Universal Robots PolyScope program: taskboard_belt_v7.urp

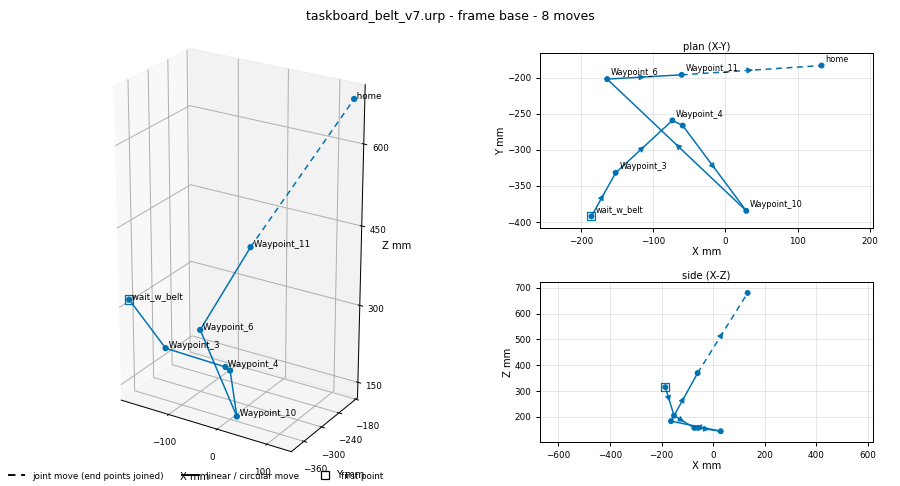
[picture p0: tool path of taskboard_belt_v7.urp in frame base, 8 of 9 moves have a stored position in this frame; points joined in program order, loops and branches not executed]
Program taskboard_belt_v7 (installation=default directory=/programs/wrs2020 createdIn=5.6.0.90886 lastSavedIn=5.9.1.1031110 robotSerialNumber=20205500180)
Calibrated DH parameters: a=[0, -0.425, -0.3922, 0, 0, 0]; d=[0.1625, 0, 0, 0.1333, 0.0997, 0.0996]; alpha=[1.570796, 0, 0, 1.570796, -1.570796, 0]; deltaTheta=[0, 0, 0, 0, 0, 0]
Robot Program (runOnlyOnce=true)
  MoveJ speed 60 deg/s, acceleration 80 deg/s^2 (useActiveTCP=true) feature=Base
    currentpose := get_actual_joint_positions()
    Waypoint Waypoint (Variable): variable=currentpose
  SuppressedNode
    Folder pick blind
      MoveJ speed 120 deg/s, acceleration 120 deg/s^2 (useActiveTCP=false) tcp=TCP; feature=Base
        Waypoint home: TCP in base x=132.399 y=-179.474 z=460.725 mm, rx=-0.0051 ry=-3.1414 rz=-0.0307 rad; joints [89.952, -120.316, 80.22, -48.701, -89.95, -0.003] deg; TCP offset x=0 y=0 z=220 mm, rx=0 ry=0 rz=0 rad
        Waypoint Waypoint_12: TCP in base x=-118.553 y=-294.346 z=577.587 mm, rx=1.3176 ry=2.7241 rz=-0.2718 rad; joints [40.024, -118.444, 99.589, -78.038, -80.282, 2.128] deg
      URCap Gripper (Robotiq_Grippers, Robotiq Inc.) dataModel(position=48.23529411764706, force=100.0, speed=100.0, positionInDouble=48.23529411764706, forceInDouble=100.0, speedInDouble=100.0, slaveIds=[9], blocking=true)
      MoveJ speed 120 deg/s, acceleration 100 deg/s^2 (useActiveTCP=false) tcp=TCP; feature=Base
        Waypoint Waypoint_1: TCP in base x=-147.509 y=-481.576 z=322.425 mm, rx=-2.2532 ry=2.177 rz=0.038 rad; joints [57.916, -85.82, 110.34, -113.684, -91.081, -124] deg; TCP offset x=0 y=0 z=0 mm, rx=0 ry=0 rz=0 rad
        MoveL speed 100 mm/s, acceleration 1200 mm/s^2 (useActiveTCP=false) tcp=TCP; feature=Base
          Waypoint Waypoint_2: TCP in base x=-147.509 y=-481.576 z=273.212 mm, rx=2.2507 ry=-2.1796 rz=-0.0127 rad; joints [57.763, -82.536, 115.155, -122.915, -90.37, -124] deg; TCP offset x=0 y=0 z=0 mm, rx=0 ry=0 rz=0 rad
      URCap Gripper (Robotiq_Grippers, Robotiq Inc.) dataModel(position=100.0, force=100.0, speed=100.0, positionInDouble=100.0, forceInDouble=100.0, speedInDouble=100.0, slaveIds=[9], blocking=true)
      MoveL speed 250 mm/s, acceleration 1200 mm/s^2 (useActiveTCP=true) feature=Base
        MoveDirectionNode (selectedDirection=ZPlus)
          Until DISTANCE (allowActions=false deceleration=3 distanceNodeType=STOP) Distance=0.1; motionParameters(blendRadius=0)
  MoveL speed 800 mm/s, acceleration 400 mm/s^2 (useActiveTCP=false) tcp=TCP; feature=Base
    SuppressedNode
      Waypoint above_tray: motionParameters(blendRadius=0.05); TCP in base x=-172.311 y=-492.624 z=406.821 mm, rx=2.0826 ry=-2.3042 rz=0.0252 rad; joints [55.84, -87.577, 100.035, -104.661, -89.581, -118.368] deg
    Waypoint wait_w_belt: TCP in base x=-185.572 y=-392.078 z=315.254 mm, rx=-1.4441 ry=1.9502 rz=-1.0486 rad; joints [37.028, -91.796, 114.934, -76.388, -46.414, -141.19] deg
  Popup Message (haltProgram=false message=start sequence together with b_bot (simultaneous start) inputType=Text)
  MoveL speed 500 mm/s, acceleration 1200 mm/s^2 (useActiveTCP=false) tcp=TCP; feature=Base
    SuppressedNode
      Waypoint Waypoint_5: TCP in base x=-173.43 y=-369.039 z=261.712 mm, rx=-1.282 ry=1.8047 rz=-1.1483 rad; joints [34.616, -88.409, 119.828, -68.558, -43.225, -150.47] deg
    Waypoint Waypoint_3: motionParameters(blendRadius=0.05); TCP in base x=-152.025 y=-331.758 z=204.759 mm, rx=-0.9043 ry=1.7298 rz=-1.6658 rad; joints [27.571, -85.137, 129.926, -53.568, -24.794, -175.111] deg
    Waypoint Waypoint_4: motionParameters(blendRadius=0.01); TCP in base x=-73.392 y=-259.129 z=157.442 mm, rx=-0.7441 ry=1.8696 rz=-1.7976 rad; joints [17.552, -96.937, 152.26, -63.92, -23.073, -175.094] deg
    Waypoint Waypoint_9: TCP in base x=-59.125 y=-266.29 z=157.434 mm, rx=-0.7441 ry=1.8696 rz=-1.7976 rad; joints [21.298, -97.571, 152.76, -64.841, -19.306, -173.924] deg
    SuppressedNode
      Waypoint Waypoint_7: TCP in base x=-93.501 y=-273.032 z=162.831 mm, rx=-0.9044 ry=1.7298 rz=-1.6658 rad; joints [21.869, -90.172, 144.622, -61.38, -30.363, -177.16] deg
  Wait Sleep waitTime=10
  URCap Gripper (Robotiq_Grippers, Robotiq Inc.) dataModel(position=80.3921568627451, force=0.0, speed=0.0, positionInDouble=80.3921568627451, forceInDouble=0.0, speedInDouble=0.0, slaveIds=[9], blocking=true)
  MoveL speed 800 mm/s, acceleration 400 mm/s^2 (useActiveTCP=false) tcp=gripper_140_tip; feature=Base
    Waypoint Waypoint_10: motionParameters(blendRadius=0.01); TCP in base x=28.985 y=-384.447 z=144.54 mm, rx=-0.9363 ry=1.6881 rz=-1.6362 rad; joints [15.25, -83.917, 139.246, -60.571, -39.887, -178.984] deg; TCP offset x=0 y=0 z=220 mm, rx=0 ry=0 rz=0 rad
    Waypoint Waypoint_6: motionParameters(blendRadius=0.04); TCP in base x=-163.794 y=-201.931 z=183.502 mm, rx=0.6153 ry=-3.0585 rz=0.0824 rad; joints [15.825, -132.373, 128.918, -87.968, -87.075, -96.888] deg
    Waypoint Waypoint_11: TCP in base x=-60.571 y=-196.005 z=369.833 mm, rx=-0.0012 ry=3.1177 rz=0.0003 rad; joints [30.867, -130.317, 98.83, -57.33, -89.307, -59.184] deg
  MoveJ speed 180 deg/s, acceleration 120 deg/s^2 (useActiveTCP=false) tcp=TCP; feature=Base
    Waypoint home: TCP in base x=133.239 y=-183.129 z=680.368 mm, rx=0.0012 ry=3.1406 rz=0.0327 rad; joints [89.956, -120.321, 80.215, -48.702, -89.954, -0.002] deg
